CASE ABB OF
	0:
		IF mxEnable AND NOT CommData.mxABBExecuting THEN
			ABB:=10;
		END_IF
	10:
		IF CommData.mxRobotOnline THEN
			ABB:=100;
			ELSE
			ABB:=200;
		END_IF
	100:
		mxExecuting:=TRUE;
		CommData.maOrderMaker[1] := 2;
		CommData.maOrderMaker[2] := 0;
		CommData.maOrderMaker[3] := 0;
		CommData.maOrderMaker[4] := 0;
		CommData.maOrderMaker[5] := 0;
		CommData.maOrderMaker[6] := 0;
		CommData.qwOrderRobot:=200000;
		ABB:=101;
	101:
		IF CommData.qwOrderRobot > 0 THEN
			CommData.qxPLCStrobe:=TRUE;
			ABB:=102;
		END_IF
	102:
		IF CommData.ixRobotStrobe THEN
			IF CommData.iwReplyRobot = CommData.qwOrderRobot+1 THEN
				CommData.qwOrderRobot:=0;
				CommData.maOrderMaker[1] := 0;
				CommData.maOrderMaker[2] := 0;
				CommData.maOrderMaker[3] := 0;
				CommData.maOrderMaker[4] := 0;
				CommData.maOrderMaker[5] := 0;
				CommData.maOrderMaker[6] := 0;
				CommData.qxPLCStrobe:=FALSE;
				ABB:=103;
			ELSE
				ABB:=1000;
			END_IF
		END_IF
	103:
		IF NOT CommData.ixRobotStrobe THEN
			IF CommData.iwReplyRobot = 0 THEN
				ABB:=104;
			ELSE
				ABB:=1000;
			END_IF
		END_IF
	104:
		IF CommData.ixRobotStrobe THEN
			IF CommData.iwProgressRobot = 90 THEN
				CommData.qxPLCStrobe:=TRUE;
				ABB:=105;
			END_IF
			IF CommData.iwProgressRobot = 1000 THEN
				CommData.qxPLCStrobe:=TRUE;
				ABB:=1000;
			END_IF
		END_IF	
	105:
		IF  NOT CommData.ixRobotStrobe AND CommData.iwProgressRobot = 0 THEN
			CommData.qxPLCStrobe:=FALSE;
			ABB:=201;
		END_IF
		
	200:
		CommData.mwABBPosXaxis:=CommData.ABBPostions.AGVPOShome.X;
		CommData.mwABBPosYaxis:=CommData.ABBPostions.AGVPOShome.Y;
		mxExecuting:=TRUE;
		CommData.mxStartABB:=TRUE;
		IF CommData.mwXaxis = CommData.ABBPostions.AGVPOShome.X AND CommData.mwYaxis = CommData.ABBPostions.AGVPOShome.Y THEN
			ABB:=201;
		ELSIF gvl.ixEmergencyStop THEN
			ABB:=1000;
		END_IF
	201:
		mxExecuting:=FALSE;
		CommData.mxStartABB:=FALSE;
		mxDone:=TRUE;
		IF NOT mxEnable THEN
			mxDone:=FALSE;
			ABB:=0;
		END_IF
	1000:
		mxError:=TRUE;
		mxExecuting:=FALSE;
		CommData.mxStartABB:=FALSE;
		IF NOT mxEnable THEN
			mxError:=FALSE;
			mxDone:=FALSE;
			ABB:=0;
		END_IF
END_CASE



IF gvl.ixEmergencyStop THEN
	ABB:=1000;
END_IF

END_FUNCTION_BLOCK

// ---- ABBControl/ABBPickLeaveContainerAGV.TcPOU
FUNCTION_BLOCK ABBPickLeaveContainerAGV
VAR_INPUT
	mxEnable: BOOL;
	mxPick: BOOL;
END_VAR
VAR_OUTPUT
	mxDone:BOOL;
	mxExecuting: BOOL;
	mxError: BOOL;
END_VAR
VAR
	ABB: INT;
	mwordernumber: DINT;
END_VAR

CASE ABB OF
	0:
		IF mxEnable AND NOT CommData.mxABBExecuting THEN
			ABB:=10;
		END_IF
	10:
		IF CommData.mxRobotOnline THEN
			ABB:=100;
			ELSE
			ABB:=200;
		END_IF
	100:
		IF CommData.msRobotLastPos = 'AGV' THEN
			ABB:=101;
		ELSE
			ABB:=1000;
		END_IF
	101:
		mxExecuting:=TRUE;
		CommData.maOrderMaker[1] := 4;
		CommData.maOrderMaker[3] := 0;
		CommData.maOrderMaker[4] := 0;
		CommData.maOrderMaker[5] := 0;
		CommData.maOrderMaker[6] := 0;
		ABB:=102;
	102:
		IF mxPick THEN
			CommData.maOrderMaker[2] := 1;
			ABB:=103;
		ELSIF NOT mxPick THEN
			CommData.maOrderMaker[2] := 0;
			ABB:=103;
		END_IF
	103:
		mwordernumber:=CommData.maOrderMaker[1];
			mwordernumber:=mwordernumber*10;
			abb:=1151;
	1151:
			mwordernumber:=mwordernumber+CommData.maOrderMaker[2];
			abb:=1152;
	1152:
			mwordernumber:=mwordernumber*10;
			abb:=1153;
	1153:
			mwordernumber:=mwordernumber+CommData.maOrderMaker[3];
			abb:=1154;
	1154:
			mwordernumber:=mwordernumber*10;
			abb:=1155;
	1155:
			mwordernumber:=mwordernumber+CommData.maOrderMaker[4];
			abb:=1156;
	1156:
			mwordernumber:=mwordernumber*10;
			abb:=1157;
	1157:
			mwordernumber:=mwordernumber+CommData.maOrderMaker[5];
			abb:=1158;
	1158:
			mwordernumber:=mwordernumber*10;
			abb:=1159;
	1159:
			mwordernumber:=mwordernumber+CommData.maOrderMaker[6];
			ABB:=1160;
	1160:
		CommData.qwOrderRobot:=mwordernumber;
		ABB:=104;
	104:
		IF CommData.qwOrderRobot > 0 THEN
			CommData.qxPLCStrobe:=TRUE;
			ABB:=105;
		END_IF
	105:
		IF CommData.ixRobotStrobe THEN
			IF CommData.iwReplyRobot = CommData.qwOrderRobot+1 THEN
				CommData.qwOrderRobot:=0;
				mwordernumber:=0;
				CommData.qxPLCStrobe:=FALSE;
				ABB:=106;
			ELSE
				ABB:=1000;
			END_IF
		END_IF
	106:
		IF NOT CommData.ixRobotStrobe THEN
			IF CommData.iwReplyRobot = 0 THEN
				ABB:=107;
			ELSE
				ABB:=1000;
			END_IF
		END_IF
	107:
		IF CommData.ixRobotStrobe THEN
			IF CommData.iwProgressRobot = 90 THEN
				CommData.qxPLCStrobe:=TRUE;
				ABB:=108;
			END_IF
			IF CommData.iwProgressRobot = 1000 THEN
				CommData.qxPLCStrobe:=TRUE;
				ABB:=1000;
			END_IF
		END_IF
	108:
		IF  NOT CommData.ixRobotStrobe AND CommData.iwProgressRobot = 0 THEN
			CommData.qxPLCStrobe:=FALSE;
			ABB:=202;
		END_IF
		
		
		
	200:
		mxExecuting:=TRUE;
		IF CommData.mwXaxis = CommData.ABBPostions.AGVPOShome.X AND CommData.mwYaxis = CommData.ABBPostions.AGVPOShome.Y THEN
			ABB:=201;
		ELSE
			ABB:=1000;
		END_IF
	201:
		IF mxpick THEN
			IF NOT CommData.mxGripper THEN
				CommData.mxGripper:=TRUE;
				ABB:=202;
			ELSE
				ABB:=1000;
			END_IF
		ELSIF NOT mxPick THEN
			IF CommData.mxGripper THEN
				CommData.mxGripper:=FALSE;
				ABB:=202;
			ELSE
				ABB:=1000;
			END_IF
		END_IF
	202:
		mxExecuting:=FALSE;
		mxDone:=TRUE;
		IF NOT mxEnable THEN
			mxError:=FALSE;
			mxDone:=FALSE;
			ABB:=0;
		END_IF
	1000:
		mxError:=TRUE;
		mxExecuting:=FALSE;
		IF NOT mxEnable THEN
			mxError:=FALSE;
			mxDone:=FALSE;
			ABB:=0;
		END_IF
END_CASE





IF gvl.ixEmergencyStop THEN
	ABB:=1000;
END_IF

END_FUNCTION_BLOCK

// ---- ABBControl/ABBScanContainer.TcPOU
FUNCTION_BLOCK ABBScanContainer
VAR_INPUT
	mxEnable: BOOL;
	mwPartno: INT;
END_VAR
VAR_OUTPUT
	mxDone: BOOL;
	mxExecuting: BOOL;
	mxRobotatScanPos:BOOL;
	mxError: BOOL;
END_VAR
VAR
	ABB: INT;
	mxWaitingforsensorinput: BOOL;
	mwordernumber: DINT;
END_VAR

CASE ABB OF
		0:
			IF mxEnable AND NOT CommData.mxABBExecuting THEN
				ABB:=10;
			END_IF
		10:
			IF CommData.mxRobotOnline THEN
			ABB:=100;
			ELSE
			ABB:=200;
		END_IF
		100:
			IF CommData.msRobotLastPos = 'Table' THEN
				ABB:=101;
			ELSE
				ABB:=1000;
			END_IF
		101:
			mxExecuting:=TRUE;
			CommData.maOrderMaker[1] := 7;
			CommData.maOrderMaker[2] := 0;
			CommData.maOrderMaker[3] := 0;
			CommData.maOrderMaker[4] := 0;
			CommData.maOrderMaker[6] := 0;
			ABB:=102;
		102:
			IF mwPartno = 1 OR mwPartno = 2 OR mwPartno = 3 THEN
				CommData.maOrderMaker[5] := mwPartno;
				ABB:=103;
			ELSE
					ABB:=1000;//Error
			END_IF
		103:
			mwordernumber:=CommData.maOrderMaker[1];
				mwordernumber:=mwordernumber*10;
				abb:=1151;
		1151:
				mwordernumber:=mwordernumber+CommData.maOrderMaker[2];
				abb:=1152;
		1152:
			mwordernumber:=mwordernumber*10;
				abb:=1153;
		1153:
				mwordernumber:=mwordernumber+CommData.maOrderMaker[3];
				abb:=1154;
		1154:
				mwordernumber:=mwordernumber*10;
				abb:=1155;
		1155:
				mwordernumber:=mwordernumber+CommData.maOrderMaker[4];
				abb:=1156;
		1156:
				mwordernumber:=mwordernumber*10;
				abb:=1157;
		1157:
				mwordernumber:=mwordernumber+CommData.maOrderMaker[5];
				abb:=1158;
		1158:
				mwordernumber:=mwordernumber*10;
				abb:=1159;
		1159:
				mwordernumber:=mwordernumber+CommData.maOrderMaker[6];
				ABB:=1160;
		1160:
			CommData.qwOrderRobot:=mwordernumber;
			ABB:=104;
		104:
			IF CommData.qwOrderRobot > 0 THEN
				CommData.qxPLCStrobe:=TRUE;
				ABB:=105;
			END_IF
		105:
			IF CommData.ixRobotStrobe THEN
				IF CommData.iwReplyRobot = CommData.qwOrderRobot+1 THEN
					CommData.qwOrderRobot:=0;
					mwordernumber:=0;
					CommData.qxPLCStrobe:=FALSE;
					ABB:=106;
				ELSE
					ABB:=1000;
				END_IF
			END_IF
		106:
			IF NOT CommData.ixRobotStrobe THEN
				IF CommData.iwReplyRobot = 0 THEN
					ABB:=1061;
				ELSE
					ABB:=1000;
				END_IF
			END_IF
		1061:
			IF CommData.iwProgressRobot = 50 THEN
				mxRobotatScanPos:=TRUE;
				ABB:=107;
			END_IF
		107:
			IF CommData.ixRobotStrobe THEN
				mxRobotatScanPos:=FALSE;
				IF CommData.iwProgressRobot = 90 THEN
					CommData.qxPLCStrobe:=TRUE;
					ABB:=108;
				END_IF
				IF CommData.iwProgressRobot = 1000 THEN
					CommData.qxPLCStrobe:=TRUE;
					ABB:=1000;
				END_IF
			END_IF
		108:
			IF  NOT CommData.ixRobotStrobe AND CommData.iwProgressRobot = 0 THEN
				CommData.qxPLCStrobe:=FALSE;
				ABB:=203;
			END_IF
		
		
		
		
		
		200:
			IF mwPartno = 1 OR mwPartno = 2 OR mwPartno = 3 THEN
				ABB:=201;
			ELSE
				ABB:=1000;//Error
			END_IF
		201:
			IF CommData.mwXaxis = CommData.ABBPostions.Tablehome.X AND CommData.mwYaxis = CommData.ABBPostions.Tablehome.Y THEN
				ABB:=202;
			ELSE
				ABB:=1000;
			END_IF
		202:
			mxExecuting:=TRUE;
			mxRobotatScanPos:=TRUE;
			commdata.mxWaitingforSensorinput:=TRUE;
			IF GVL.ixInductiveSensorinTool OR CommData.mxScannernoobject THEN
				ABB:=203;
			END_IF
		203:
			commdata.mxWaitingforSensorinput:=FALSE;
			mxRobotatScanPos:=FALSE;
			mxExecuting:=FALSE;
			mxDone:=TRUE;
			IF NOT mxEnable THEN
				mxDone:=FALSE;
				ABB:=0;
			END_IF
		1000:
			mxExecuting:=FALSE;
			mxError:=TRUE;
			IF NOT mxEnable THEN
				mxError:=FALSE;
				mxDone:=FALSE;
				ABB:=0;
			END_IF
END_CASE



IF gvl.ixEmergencyStop THEN
	ABB:=1000;
END_IF

END_FUNCTION_BLOCK

// ---- ABBControl/ABBGotoTable.TcPOU
FUNCTION_BLOCK ABBGotoTable
VAR_INPUT
	mxEnable: BOOL;
END_VAR
VAR_OUTPUT
	mxDone:BOOL;
	mxExecuting: BOOL;
	mxError: BOOL;
END_VAR
VAR
	ABB: INT;
END_VAR

CASE ABB OF
	0:
		IF mxEnable AND NOT CommData.mxABBExecuting THEN
			ABB:=10;
		END_IF
	10:
		IF CommData.mxRobotOnline THEN
			ABB:=100;
		ELSE
			ABB:=200;
		END_IF
	100:
		mxExecuting:=TRUE;
		CommData.maOrderMaker[1] := 3;
		CommData.maOrderMaker[2] := 0;
		CommData.maOrderMaker[3] := 0;
		CommData.maOrderMaker[4] := 0;
		CommData.maOrderMaker[5] := 0;
		CommData.maOrderMaker[6] := 0;
		CommData.qwOrderRobot:=300000;
		ABB:=101;
	101:
		IF CommData.qwOrderRobot > 0 THEN
			CommData.qxPLCStrobe:=TRUE;
			ABB:=102;
		END_IF
	102:
		IF CommData.ixRobotStrobe THEN
			IF CommData.iwReplyRobot = CommData.qwOrderRobot+1 THEN
				CommData.qwOrderRobot:=0;
				CommData.maOrderMaker[1] := 0;
				CommData.maOrderMaker[2] := 0;
				CommData.maOrderMaker[3] := 0;
				CommData.maOrderMaker[4] := 0;
				CommData.maOrderMaker[5] := 0;
				CommData.maOrderMaker[6] := 0;
				CommData.qxPLCStrobe:=FALSE;
				ABB:=103;
			ELSE
				ABB:=1000;
			END_IF
		END_IF
	103:
		IF NOT CommData.ixRobotStrobe THEN
			IF CommData.iwReplyRobot = 0 THEN
				ABB:=104;
			ELSE
				ABB:=1000;
			END_IF
		END_IF
	104:
		IF CommData.ixRobotStrobe THEN
			IF CommData.iwProgressRobot = 90 THEN
				CommData.qxPLCStrobe:=TRUE;
				ABB:=105;
			END_IF
			IF CommData.iwProgressRobot = 1000 THEN
				CommData.qxPLCStrobe:=TRUE;
				ABB:=1000;
			END_IF
		END_IF	
	105:
		IF  NOT CommData.ixRobotStrobe AND CommData.iwProgressRobot = 0 THEN
			CommData.qxPLCStrobe:=FALSE;
			ABB:=201;
		END_IF
		
		
	200:
		CommData.mwABBPosXaxis:=CommData.ABBPostions.Tablehome.X;
		CommData.mwABBPosYaxis:=CommData.ABBPostions.Tablehome.Y;
		mxExecuting:=TRUE;
		CommData.mxStartABB:=TRUE;
		IF CommData.mwXaxis = CommData.ABBPostions.Tablehome.X AND CommData.mwYaxis = CommData.ABBPostions.Tablehome.Y THEN
			ABB:=201;
		ELSIF gvl.ixEmergencyStop THEN
			ABB:=1000;
		END_IF
	201:
		mxExecuting:=FALSE;
		CommData.mxStartABB:=FALSE;
		mxDone:=TRUE;
		IF NOT mxEnable THEN
			mxDone:=FALSE;
			ABB:=0;
		END_IF
	1000:
		mxError:=TRUE;
		mxExecuting:=FALSE;
		CommData.mxStartABB:=FALSE;
		IF NOT mxEnable THEN
			mxError:=FALSE;
			mxDone:=FALSE;
			ABB:=0;
		END_IF
END_CASE



IF gvl.ixEmergencyStop THEN
	ABB:=1000;
END_IF

END_FUNCTION_BLOCK

// ---- ABBControl/ABBAssemble.TcPOU
FUNCTION_BLOCK ABBAssemble
VAR_INPUT
	mxEnable: BOOL;
	mwBufferID: INT;
END_VAR
VAR_OUTPUT
	mxDone: BOOL;
	mxExecuting: BOOL;
	mxError: BOOL;
END_VAR
VAR
	ABB: INT;
	mwPlatecount: INT;
	mwordernumber: DINT;
END_VAR
VAR_INPUT
	mwAssemblePartno: INT;
END_VAR

CASE ABB OF
	0:
		IF mxEnable AND NOT CommData.mxABBExecuting THEN
			ABB:=10;
		END_IF
	10:
		IF CommData.mxRobotOnline THEN
			ABB:=11;
			ELSE
			ABB:=12;
		END_IF
	11:
		IF CommData.msRobotLastPos = 'Table' AND gvl.BufferProducts.Storage1.Quatity <> 0 AND gvl.BufferProducts.Storage2.Quatity <> 0 AND gvl.BufferProducts.Storage3.Quatity <> 0 THEN
			ABB:=111;
		ELSE
			ABB:=1000;
		END_IF
	111:
		mxExecuting:=TRUE;
		CommData.maOrderMaker[1] := 8;
		CommData.maOrderMaker[2] := 0;
		IF mwAssemblePartno =3 THEN
			abb:=112;
		ELSIF mwAssemblePartno =2 THEN
			abb:=113;
		ELSIF mwAssemblePartno =1 THEN
			abb:=114;
		END_IF	
	112:
		IF mwBufferID = 1 THEN
				CommData.maOrderMaker[3]:=mwBufferID;
				CommData.maOrderMaker[4]:=gvl.BufferProducts.Storage1.Quatity;
				CommData.maOrderMaker[5]:=mwAssemblePartno;
				CommData.maOrderMaker[6]:=0;
				abb:=115;
			ELSIF mwBufferID = 2 THEN
				CommData.maOrderMaker[3]:=mwBufferID;
				CommData.maOrderMaker[4]:=gvl.BufferProducts.Storage2.Quatity;
				CommData.maOrderMaker[5]:=mwAssemblePartno;
				CommData.maOrderMaker[6]:=0;
				abb:=115;
			ELSIF mwBufferID = 3 THEN
				CommData.maOrderMaker[3]:=mwBufferID;
				CommData.maOrderMaker[4]:=gvl.BufferProducts.Storage3.Quatity;
				CommData.maOrderMaker[5]:=mwAssemblePartno;
				CommData.maOrderMaker[6]:=0;
				abb:=115;
			ELSE
				ABB:=1000;
			END_IF
	113:
		IF mwBufferID = 1 THEN
				CommData.maOrderMaker[3]:=mwBufferID;
				CommData.maOrderMaker[4]:=gvl.BufferProducts.Storage1.Quatity;
				CommData.maOrderMaker[5]:=mwAssemblePartno;
				CommData.maOrderMaker[6]:=0;
				abb:=115;
			ELSIF mwBufferID = 2 THEN
				CommData.maOrderMaker[3]:=mwBufferID;
				CommData.maOrderMaker[4]:=gvl.BufferProducts.Storage2.Quatity;
				CommData.maOrderMaker[5]:=mwAssemblePartno;
				CommData.maOrderMaker[6]:=0;
				abb:=115;
			ELSIF mwBufferID = 3 THEN
				CommData.maOrderMaker[3]:=mwBufferID;
				CommData.maOrderMaker[4]:=gvl.BufferProducts.Storage3.Quatity;
				CommData.maOrderMaker[5]:=mwAssemblePartno;
				CommData.maOrderMaker[6]:=0;
				abb:=115;
			ELSE
				ABB:=1000;
			END_IF
	114:
		IF gvl.BufferProducts.Storage3.Quatity =2 THEN
			mwPlatecount:=6;
		ELSIF gvl.BufferProducts.Storage3.Quatity =1 THEN
			mwPlatecount:=5;
		END_IF
		IF mwBufferID = 1 THEN
				IF gvl.BufferProducts.Storage1.Quatity =2 THEN
					mwPlatecount:=6;
					abb:=1141;
				ELSIF gvl.BufferProducts.Storage1.Quatity =1 THEN
					mwPlatecount:=5;
					abb:=1141;
				END_IF
		ELSIF mwBufferID = 2 THEN
				IF gvl.BufferProducts.Storage2.Quatity =2 THEN
					mwPlatecount:=6;
					abb:=1141;
				ELSIF gvl.BufferProducts.Storage2.Quatity =1 THEN
					mwPlatecount:=5;
					abb:=1141;
				END_IF
		ELSIF mwBufferID = 3 THEN
				IF gvl.BufferProducts.Storage3.Quatity =2 THEN
					mwPlatecount:=6;
					abb:=1141;
				ELSIF gvl.BufferProducts.Storage3.Quatity =1 THEN
					mwPlatecount:=5;
					abb:=1141;
				END_IF
			ELSE
				ABB:=1000;
			END_IF
	1141:
		CommData.maOrderMaker[3]:=mwBufferID;
		CommData.maOrderMaker[4]:=mwPlatecount;
		CommData.maOrderMaker[5]:=mwAssemblePartno;
		CommData.maOrderMaker[6]:=0;
		abb:=115;
	115:
		IF CommData.maOrderMaker[1]=8 THEN
			mwordernumber:=CommData.maOrderMaker[1];
			mwordernumber:=mwordernumber*10;
			abb:=1151;
		END_IF
	1151:
			mwordernumber:=mwordernumber+CommData.maOrderMaker[2];
			abb:=1152;
	1152:
			mwordernumber:=mwordernumber*10;
			abb:=1153;
	1153:
			mwordernumber:=mwordernumber+CommData.maOrderMaker[3];
			abb:=1154;
	1154:
			mwordernumber:=mwordernumber*10;
			abb:=1155;
	1155:
			mwordernumber:=mwordernumber+CommData.maOrderMaker[4];
			abb:=1156;
	1156:
			mwordernumber:=mwordernumber*10;
			abb:=1157;
	1157:
			mwordernumber:=mwordernumber+CommData.maOrderMaker[5];
			abb:=1158;
	1158:
			mwordernumber:=mwordernumber*10;
			abb:=1159;
	1159:
			mwordernumber:=mwordernumber+CommData.maOrderMaker[6];
			ABB:=116;

	116:
		CommData.qwOrderRobot:=mwordernumber;
		ABB:=117;
	117:
		IF CommData.qwOrderRobot > 0 THEN
			CommData.qxPLCStrobe:=TRUE;
			ABB:=118;
		END_IF
	118:
		IF CommData.ixRobotStrobe THEN
			IF CommData.iwReplyRobot = CommData.qwOrderRobot+1 THEN
				CommData.qwOrderRobot:=0;
				mwordernumber:=0;
				CommData.qxPLCStrobe:=FALSE;
				ABB:=119;
			ELSE
				ABB:=1000;
			END_IF
		END_IF
	119:
		IF NOT CommData.ixRobotStrobe THEN
			IF CommData.iwReplyRobot = 0 THEN
				ABB:=120;
			ELSE
				ABB:=1000;
			END_IF
		END_IF
	120:
		IF CommData.ixRobotStrobe THEN
			IF CommData.iwProgressRobot = 90 THEN
				CommData.qxPLCStrobe:=TRUE;
				ABB:=121;
			END_IF
			IF CommData.iwProgressRobot = 1000 THEN
				CommData.qxPLCStrobe:=TRUE;
				ABB:=1000;
			END_IF
		END_IF
	121:
		IF  NOT CommData.ixRobotStrobe AND CommData.iwProgressRobot = 0 THEN
			CommData.qxPLCStrobe:=FALSE;
			ABB:=73;
		END_IF
	12:
		IF CommData.mwXaxis = CommData.ABBPostions.Tablehome.X AND CommData.mwYaxis = CommData.ABBPostions.Tablehome.Y THEN
			ABB:=20;
		ELSE
			ABB:=1000;
		END_IF
	20:
		mxExecuting:=TRUE;
		CommData.mwABBPosXaxis:=CommData.ABBPostions.Bufferhome.X;
		CommData.mwABBPosYaxis:=CommData.ABBPostions.Bufferhome.Y;
		CommData.mxStartABB:=TRUE;
		IF CommData.mwXaxis = CommData.ABBPostions.Bufferhome.X AND CommData.mwYaxis = CommData.ABBPostions.Bufferhome.Y THEN
			CommData.mxStartABB:=FALSE;
			ABB:=30;
		ELSIF gvl.ixEmergencyStop THEN
			ABB:=1000;
		END_IF
	30:
		IF mwBufferID = 1 THEN
			ABB:=40;
		ELSIF mwBufferID = 2 THEN
			ABB:=50;
		ELSIF mwBufferID = 3 THEN
			ABB:=60;
		ELSE
			ABB:=1000;//Error
		END_IF
	40:
		CommData.mwABBPosXaxis:=CommData.ABBPostions.Storage1.X;
		CommData.mwABBPosYaxis:=CommData.ABBPostions.Storage1.Y;
		CommData.mxStartABB:=TRUE;
		IF CommData.mwXaxis = CommData.ABBPostions.Storage1.X AND CommData.mwYaxis = CommData.ABBPostions.Storage1.Y THEN
			CommData.mxStartABB:=FALSE;
			ABB:=70;
		END_IF
	50:
		CommData.mwABBPosXaxis:=CommData.ABBPostions.Storage2.X;
		CommData.mwABBPosYaxis:=CommData.ABBPostions.Storage2.Y;
		CommData.mxStartABB:=TRUE;
		IF CommData.mwXaxis = CommData.ABBPostions.Storage2.X AND CommData.mwYaxis = CommData.ABBPostions.Storage2.Y THEN
			CommData.mxStartABB:=FALSE;
			ABB:=70;
		END_IF
	60:
		CommData.mwABBPosXaxis:=CommData.ABBPostions.Storage3.X;
		CommData.mwABBPosYaxis:=CommData.ABBPostions.Storage3.Y;
		CommData.mxStartABB:=TRUE;
		IF CommData.mwXaxis = CommData.ABBPostions.Storage3.X AND CommData.mwYaxis = CommData.ABBPostions.Storage3.Y THEN
			CommData.mxStartABB:=FALSE;
			ABB:=70;
		END_IF
		
		
		
	70:
		IF NOT CommData.mxABBExecuting THEN
			IF NOT CommData.mxGripper THEN
				CommData.mxGripper:=TRUE;
				ABB:=71;
			ELSE
				ABB:=1000;
			END_IF
		END_IF
	71:
		CommData.mwABBPosXaxis:=CommData.ABBPostions.Tablehome.X;
		CommData.mwABBPosYaxis:=CommData.ABBPostions.Tablehome.Y;
		CommData.mxStartABB:=TRUE;
		IF CommData.mwXaxis = CommData.ABBPostions.Tablehome.X AND CommData.mwYaxis = CommData.ABBPostions.Tablehome.Y THEN
			CommData.mxStartABB:=FALSE;
			ABB:=72;
		END_IF
	72:
		IF CommData.mxGripper THEN
			CommData.mxGripper:=FALSE;
			ABB:=73;
		ELSE
			ABB:=40;
		END_IF
	73:
		mxExecuting:=FALSE;
		mxDone:=TRUE;
		IF NOT mxEnable THEN
			mxError:=FALSE;
			mxDone:=FALSE;
			ABB:=0;
		END_IF
	1000:
		mxError:=TRUE;
		mxExecuting:=FALSE;
		CommData.mxStartABB:=FALSE;
		IF NOT mxEnable THEN
			mxError:=FALSE;
			mxDone:=FALSE;
			ABB:=0;
		END_IF
END_CASE


IF gvl.ixEmergencyStop THEN
	ABB:=1000;
END_IF

END_FUNCTION_BLOCK

// ---- ABBControl/ABBPickLeaveContaineronTable.TcPOU
FUNCTION_BLOCK ABBPickLeaveContaineronTable
VAR_INPUT
	mxEnable: BOOL;
	mxPick: BOOL;
END_VAR
VAR_OUTPUT
	mxDone:BOOL;
	mxExecuting: BOOL;
	mxError: BOOL;
END_VAR
VAR
	ABB: INT;
	mwordernumber: DINT;
END_VAR

CASE ABB OF
	0:
		IF mxEnable AND NOT CommData.mxABBExecuting THEN
			ABB:=10;
		END_IF
	10:
		IF CommData.mxRobotOnline THEN
			ABB:=100;
			ELSE
			ABB:=200;
		END_IF
	100:
		IF CommData.msRobotLastPos = 'Table' THEN
			ABB:=101;
		ELSE
			ABB:=1000;
		END_IF
	101:
		mxExecuting:=TRUE;
		CommData.maOrderMaker[1] := 5;
		CommData.maOrderMaker[3] := 0;
		CommData.maOrderMaker[4] := 0;
		CommData.maOrderMaker[5] := 0;
		CommData.maOrderMaker[6] := 0;
		ABB:=102;
	102:
		IF mxPick THEN
			CommData.maOrderMaker[2] := 1;
			ABB:=103;
		ELSIF NOT mxPick THEN
			CommData.maOrderMaker[2] := 0;
			ABB:=103;
		END_IF
	103:
		mwordernumber:=CommData.maOrderMaker[1];
			mwordernumber:=mwordernumber*10;
			abb:=1151;
	1151:
			mwordernumber:=mwordernumber+CommData.maOrderMaker[2];
			abb:=1152;
	1152:
			mwordernumber:=mwordernumber*10;
			abb:=1153;
	1153:
			mwordernumber:=mwordernumber+CommData.maOrderMaker[3];
			abb:=1154;
	1154:
			mwordernumber:=mwordernumber*10;
			abb:=1155;
	1155:
			mwordernumber:=mwordernumber+CommData.maOrderMaker[4];
			abb:=1156;
	1156:
			mwordernumber:=mwordernumber*10;
			abb:=1157;
	1157:
			mwordernumber:=mwordernumber+CommData.maOrderMaker[5];
			abb:=1158;
	1158:
			mwordernumber:=mwordernumber*10;
			abb:=1159;
	1159:
			mwordernumber:=mwordernumber+CommData.maOrderMaker[6];
			ABB:=1160;
	1160:
		CommData.qwOrderRobot:=mwordernumber;
		ABB:=104;
	104:
		IF CommData.qwOrderRobot > 0 THEN
			CommData.qxPLCStrobe:=TRUE;
			ABB:=105;
		END_IF
	105:
		IF CommData.ixRobotStrobe THEN
			IF CommData.iwReplyRobot = CommData.qwOrderRobot+1 THEN
				CommData.qwOrderRobot:=0;
				mwordernumber:=0;
				CommData.qxPLCStrobe:=FALSE;
				ABB:=106;
			ELSE
				ABB:=1000;
			END_IF
		END_IF
	106:
		IF NOT CommData.ixRobotStrobe THEN
			IF CommData.iwReplyRobot = 0 THEN
				ABB:=107;
			ELSE
				ABB:=1000;
			END_IF
		END_IF
	107:
		IF CommData.ixRobotStrobe THEN
			IF CommData.iwProgressRobot = 90 THEN
				CommData.qxPLCStrobe:=TRUE;
				ABB:=108;
			END_IF
			IF CommData.iwProgressRobot = 1000 THEN
				CommData.qxPLCStrobe:=TRUE;
				ABB:=1000;
			END_IF
		END_IF
	108:
		IF  NOT CommData.ixRobotStrobe AND CommData.iwProgressRobot = 0 THEN
			CommData.qxPLCStrobe:=FALSE;
			ABB:=202;
		END_IF
	

	200:
		mxExecuting:=TRUE;
		IF CommData.mwXaxis = CommData.ABBPostions.Tablehome.X AND CommData.mwYaxis = CommData.ABBPostions.Tablehome.Y THEN
			ABB:=201;
		ELSE
			mxError:=TRUE;
			ABB:=40;
		END_IF
	201:
		IF mxpick THEN
			IF NOT CommData.mxGripper THEN
				CommData.mxGripper:=TRUE;
				ABB:=202;
			ELSE
				ABB:=1000;
			END_IF
		ELSIF NOT mxPick THEN
			IF CommData.mxGripper THEN
				CommData.mxGripper:=FALSE;
				ABB:=202;
			ELSE
				ABB:=1000;
			END_IF
		END_IF
	202:
		mxExecuting:=FALSE;
		mxDone:=TRUE;
		IF NOT mxEnable THEN
			mxError:=FALSE;
			mxDone:=FALSE;
			ABB:=0;
		END_IF
	1000:  //Error State
		mxError:=TRUE;
		mxExecuting:=FALSE;
		IF NOT mxEnable THEN
			mxError:=FALSE;
			mxDone:=FALSE;
			ABB:=0;
		END_IF
END_CASE




IF gvl.ixEmergencyStop THEN
	ABB:=1000;
END_IF

END_FUNCTION_BLOCK

// ---- Automation Library/PhysicalSystemTest.TcPOU
PROGRAM PhysicalSystemTest
VAR
	ABB: INT;
	TwoSecTimer: TON;
	mxTimerStart:BOOL;
	mxTimerDone:BOOL;
END_VAR

CASE ABB OF
	0:
		IF CommData.qxPLCStrobe THEN
			ABB:=10;
		END_IF
	10:
		IF CommData.qwOrderRobot > 0 THEN
			CommData.iwReplyRobot:=CommData.qwOrderRobot+1;
			mxTimerStart:=TRUE;
			ABB:=20;
		END_IF
	20:
		IF mxTimerDone THEN
			CommData.ixRobotStrobe :=TRUE;
			mxTimerStart:=FALSE;
			ABB:=30;
		END_IF
	30:
		IF NOT CommData.qxPLCStrobe THEN
			mxTimerStart:=TRUE;
			ABB:=40;
		END_IF
	40:
		IF mxTimerDone THEN
			CommData.iwReplyRobot:=0;
			CommData.ixRobotStrobe :=FALSE;
			mxTimerStart:=FALSE;
			ABB:=50;
		END_IF
	50:
		mxTimerStart:=TRUE;
		IF mxTimerDone THEN
			mxTimerStart:=FALSE;
			CommData.iwProgressRobot:=90;
			ABB:=60;
		END_IF
	60:
		CommData.ixRobotStrobe :=TRUE;
		mxTimerStart:=TRUE;
		ABB:=70;
	70:
		IF mxTimerDone AND CommData.qxPLCStrobe THEN
			mxTimerStart:=FALSE;
			CommData.iwProgressRobot:=0;
			ABB:=80;
		END_IF
	80:
		mxTimerStart:=TRUE;
		IF mxTimerDone THEN
			mxTimerStart:=FALSE;
			CommData.ixRobotStrobe :=FALSE;
			ABB:=90;
		END_IF
	90:
		IF NOT CommData.qxPLCStrobe THEN
			ABB:=0;
		END_IF
END_CASE



TwoSecTimer(IN:= mxTimerStart, PT:= T#2S, Q=> mxTimerDone, ET=> );

END_PROGRAM

// ---- GlobalTextList.TcGTLO
TEXTLIST GlobalTextList
  153 = ' %s'
  135 = '%s'
  875 = '1'
  207 = '2'
  288 = '3'
  990 = 'ABB Error'
  910 = 'ABB Executing'
  564 = 'ABB Functions'
  615 = 'ABB Onlibe'
  693 = 'ABB Status'
  435 = 'AGV'
  139 = 'AGV at Station :'
  241 = 'AGV Pos'
  375 = 'AGV Scan Table'
  171 = 'All Buffer Check'
  575 = 'All Home Check'
  974 = 'Aseembly'
  126 = 'Assemble'
  522 = 'Assembling'
  423 = 'Auto'
  27 = 'Auto Mode'
  641 = 'Booking from IO Station  :'
  114 = 'Buffer'
  731 = 'Buffer 1'
  938 = 'Buffer 2'
  402 = 'Buffer 3'
  289 = 'Buffer Empty'
  769 = 'Buffer ID'
  25 = 'BufferID'
  512 = 'Checkbox'
  728 = 'Container'
  514 = 'Container Color'
  281 = 'Control for Station'
  685 = 'Cylinder'
  150 = 'Debug Mode'
  228 = 'DebugMode'
  379 = 'Dummy BUffer'
  698 = 'Dummy Buffer'
  390 = 'Emergency Mode'
  137 = 'Emergency Signal :'
  493 = 'Emergency Stop'
  136 = 'Error from Comm :'
  999 = 'Execute'
  93 = 'Finish Order'
  170 = 'Gabriel Sebastian'
  751 = 'Gabriel Sebastian gabriel.sebastian@hv.se'
  995 = 'Gabriel Sebastian | gabriel.sebastian@hv.se'
  701 = 'Gabriel Sebastian |gabriel.sebastian@hv.se'
  922 = 'Go to Pos'
  688 = 'Gripper Control'
  247 = 'Gripper Toggle'
  222 = 'Home'
  140 = 'Inventory Status'
  395 = 'ixAGVatStation'
  884 = 'Leave'
  498 = 'Leave at AGV'
  298 = 'Main Menu'
  319 = 'Manual'
  917 = 'Manual Controller'
  314 = 'Manual Controls'
  212 = 'Manual Mode'
  122 = 'Manual Scanning'
  792 = 'Mode Status'
  1015 = 'New AGV to Station'
  203 = 'New AGV to Station :'
  151 = 'Normal Mode'
  908 = 'Octagon'
  287 = 'OFF'
  363 = 'Offline'
  741 = 'OFFLINE'
  374 = 'ON'
  13 = 'Online'
  979 = 'ONLINE'
  174 = 'Order for Next Assembly  : %s'
  138 = 'Pallet Placed on AGV :'
  147 = 'Pallet Sensor 1  :'
  146 = 'Pallet Sensor 2  :'
  148 = 'Pallet Sensor 3  :'
  145 = 'Pallet Sensor 4  :'
  563 = 'Part'
  315 = 'Part 1'
  242 = 'Part 2'
  436 = 'Part 3'
  331 = 'Part ID'
  213 = 'PartID'
  874 = 'Pause'
  105 = 'Paused'
  339 = 'Pick'
  758 = 'Pick / Leave'
  110 = 'Plate'
  669 = 'PLC'
  646 = 'Quantity'
  196 = 'Request Generator'
  835 = 'Reset'
  166 = 'Reset ABB'
  883 = 'Reset Station'
  867 = 'Reset Task'
  556 = 'Robot'
  625 = 'Robot Position  : %s'
  881 = 'Robot Power'
  502 = 'Robot Station'
  583 = 'Scan Buffer 1'
  714 = 'Scan Buffer 2'
  354 = 'Scan Buffer 3'
  620 = 'Scan Container'
  204 = 'Scanner'
  973 = 'Scanning'
  83 = 'Send Order'
  899 = 'Sensor Reading  : %s'
  238 = 'Sensor Reading completed'
  144 = 'Sensor Signals'
  134 = 'Station ID :'
  152 = 'Station Offline'
  494 = 'Station Status  : %s'
  458 = 'Station View'
  169 = 'Stop'
  143 = 'Storage Pos 1: %s'
  141 = 'Storage Pos 2: %s'
  142 = 'Storage Pos 3: %s'
  456 = 'SubTask'
  549 = 'Table'
  266 = 'Table To AGV'
  882 = 'Task'
  229 = 'Task Section'
  309 = 'Test System'
  149 = 'Tool Sensor  :'
  886 = 'Visualization'
  127 = 'X  : %s'
  412 = 'Y  : %s'
END_TEXTLIST

// ---- VISUs/RobotStation.TcVIS
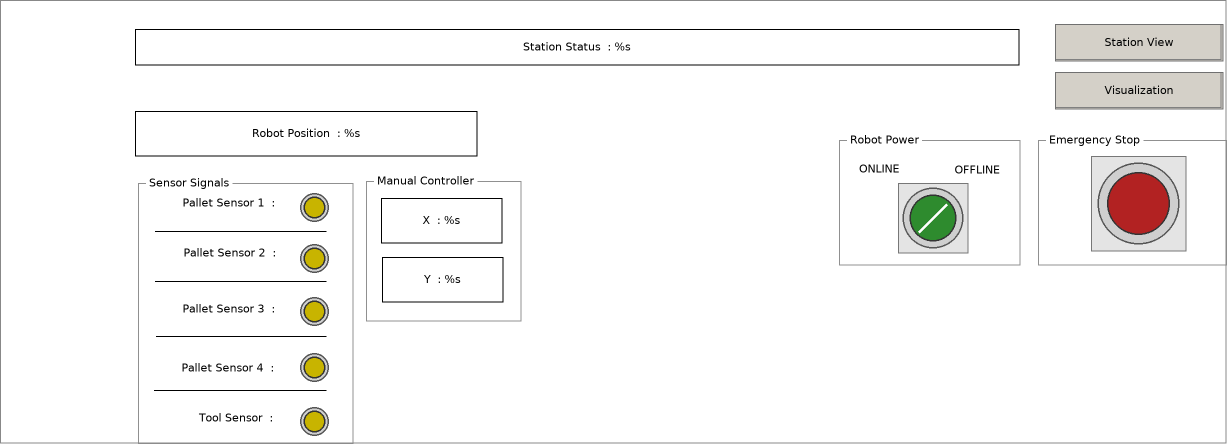
VISUALIZATION RobotStation  // 1227x444
    Rectangle (135,29 884x36), "Station Status : %s", text variable: Visualaisation_Control.mxStationStatus
    GroupBox (839,132 181x133), "Robot Power", invisible if: CommData.mxOnlineMode
        RotarySwitch (59,51 70x70), variable: CommData.mxRobotOnline, invisible if: CommData.mxOnlineMode, behaviour: TOGGLE, style: Switch-RotarySwitch-Green
        Label (11,22 59x30), "ONLINE"
        Label (106,23 65x30), "OFFLINE"
    Button (1055,72 168x37), "Visualization"
        OnMouseClick: change screen: Visualization
    GroupBox (1038,132 189x133), "Emergency Stop"
        PushSwitch (45,24 111x95), variable: GVL.ixEmergencyStop, behaviour: TOGGLE, style: Switch-PushSwitch-Red
    Rectangle (135,111 342x45), "Robot Position : %s", text variable: CommData.msRobotLastPos
    GroupBox (138,175 215x269), "Sensor Signals"
        Label (15,178 150x30), "Pallet Sensor 4 :"
        Label (17,63 150x30), "Pallet Sensor 2 :"
        Line (17,56) (188,56)
        Lamp1 (160,16 33x33), variable: GVL.ixInductiveSensor1, style: Lamp-Lamp1-Yellow
        Lamp1 (160,67 33x33), variable: GVL.ixInductiveSensor2, style: Lamp-Lamp1-Yellow
        Lamp1 (160,120 33x33), variable: GVL.ixInductiveSensor3, style: Lamp-Lamp1-Yellow
        Lamp1 (160,176 33x33), variable: GVL.ixInductiveSensor4, style: Lamp-Lamp1-Yellow
        Label (16,119 150x30), "Pallet Sensor 3 :"
        Label (23,228 150x30), "Tool Sensor :"
        Lamp1 (160,230 33x33), variable: GVL.ixInductiveSensorinTool, style: Lamp-Lamp1-Yellow
        Line (17,106) (188,106)
        Line (18,161) (188,161)
        Line (16,215) (188,215)
        Label (16,13 150x30), "Pallet Sensor 1 :"
    GroupBox (366,173 155x148), "Manual Controller"
        Rectangle (16,84 121x45), "Y : %s", text variable: CommData.mwYaxis
            OnMouseClick: write the text variable via Default
        Rectangle (15,25 121x45), "X : %s", text variable: CommData.mwXaxis
            OnMouseClick: write the text variable via Default
    Button (1055,24 168x37), "Station View"
        OnMouseClick: change screen: Station
END_VISUALIZATION

// ---- VISUs/Station.TcVIS
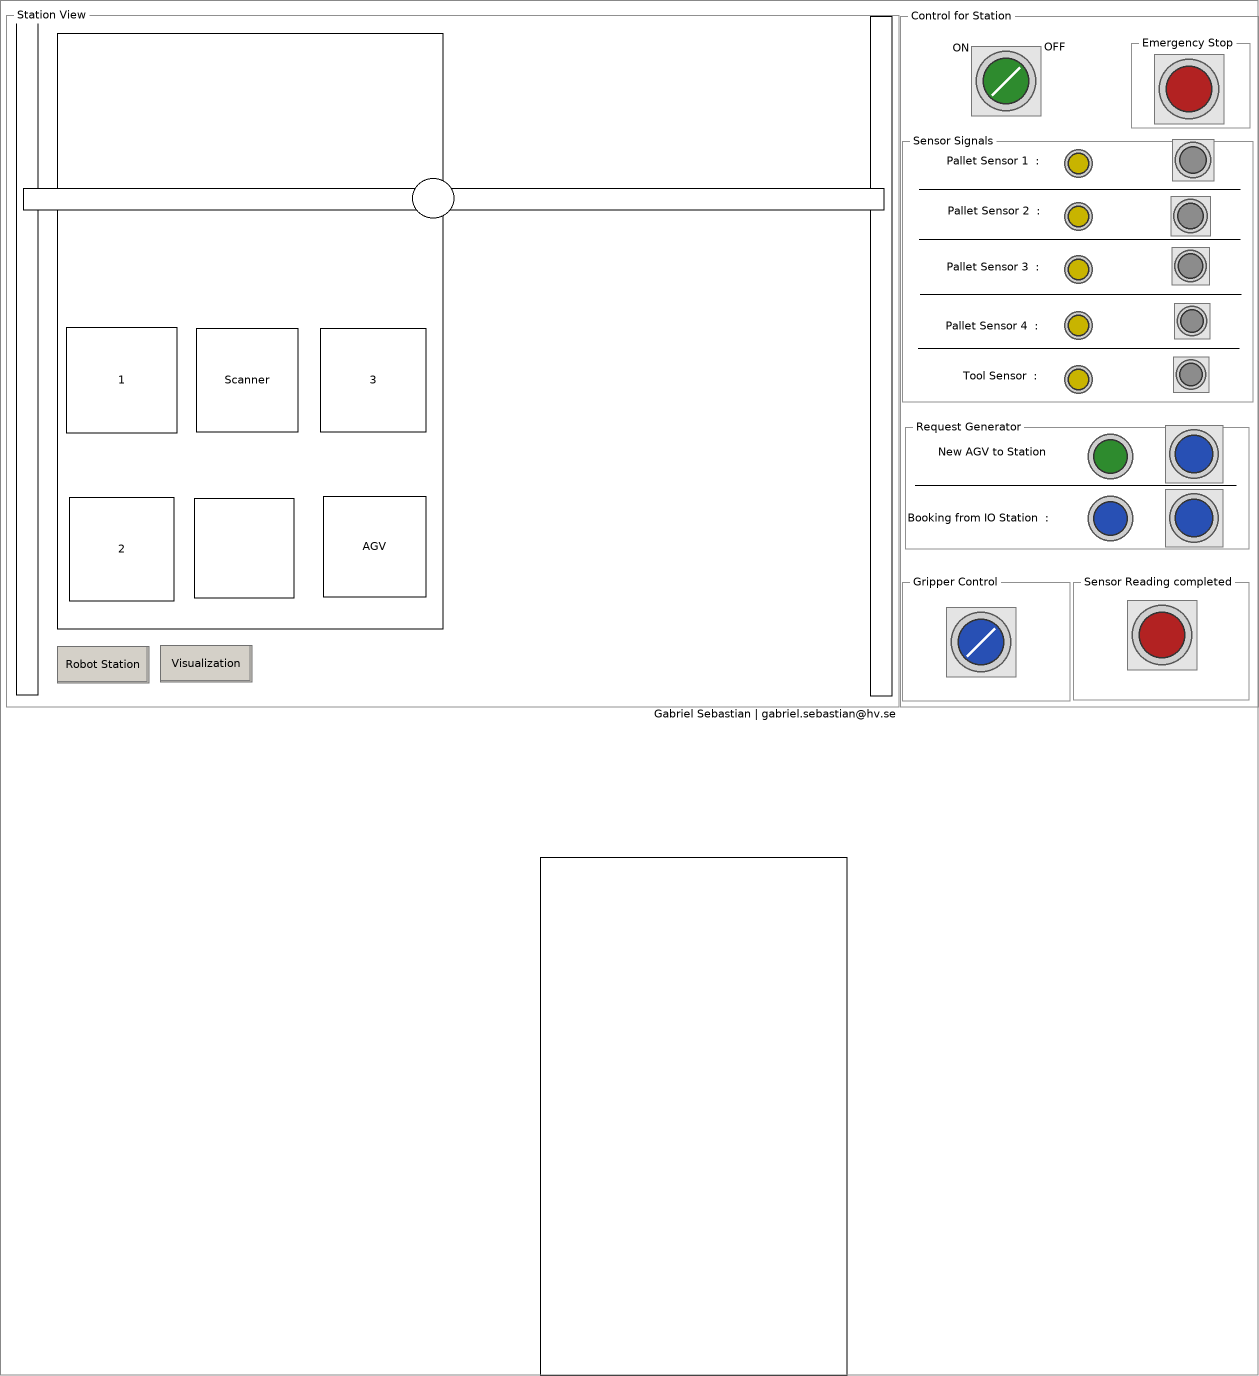
VISUALIZATION Station  // 1259x1376
    RoundedRectangle (540,857 307x519)
        p2738717112: CommData.mwCurrentAGVPOS
    Rectangle (16,15 22x680)
    GroupBox (6,7 893x700), "Station View"
        Rectangle (51,26 386x596)
        Rectangle (864,9 22x680)
        Rectangle (188,491 100x100)
        Rectangle (317,489 103x101), "AGV"
        Rectangle (190,321 102x104), "Scanner"
        Rectangle (60,320 111x106), "1"
        Rectangle (314,321 106x104), "3"
        Rectangle (63,490 105x104), "2"
        RoundedRectangle (17,181 861x22)
            p2738717112: CommData.mwYaxis
        Ellipse (406,171 42x40)
            p2738717112: CommData.mwYaxis
            p3560616238: CommData.mwXaxis
        Button (154,638 92x37), "Visualization"
            OnMouseClick: change screen: Visualization
        Button (51,639 92x37), "Robot Station"
            OnMouseClick: change screen: RobotStation
    GroupBox (900,8 359x699), "Control for Station"
        GroupBox (2,125 351x269), "Sensor Signals"
            Label (15,178 150x30), "Pallet Sensor 4 :"
            Label (17,63 150x30), "Pallet Sensor 2 :"
            Label (16,13 150x30), "Pallet Sensor 1 :"
            Line (17,56) (338,56)
            Lamp1 (160,14 33x33), variable: GVL.ixInductiveSensor1, style: Lamp-Lamp1-Yellow
            Lamp1 (160,67 33x33), variable: GVL.ixInductiveSensor2, style: Lamp-Lamp1-Yellow
            Lamp1 (160,120 33x33), variable: GVL.ixInductiveSensor3, style: Lamp-Lamp1-Yellow
            Lamp1 (160,176 33x33), variable: GVL.ixInductiveSensor4, style: Lamp-Lamp1-Yellow
            Label (16,119 150x30), "Pallet Sensor 3 :"
            Label (23,228 150x30), "Tool Sensor :"
            Lamp1 (160,230 33x33), variable: GVL.ixInductiveSensorinTool, style: Lamp-Lamp1-Yellow
            PushSwitch (266,6 50x42), variable: GVL.ixInductiveSensor1, input disabled if: CommData.mxRobotOnline, behaviour: TOGGLE, style: Switch-PushSwitch-Gray
            PushSwitch (267,63 43x40), variable: GVL.ixInductiveSensor2, input disabled if: CommData.mxRobotOnline, behaviour: TOGGLE, style: Switch-PushSwitch-Gray
            PushSwitch (269,114 39x38), variable: GVL.ixInductiveSensor3, input disabled if: CommData.mxRobotOnline, behaviour: TOGGLE, style: Switch-PushSwitch-Gray
            PushSwitch (270,170 40x36), variable: GVL.ixInductiveSensor4, input disabled if: CommData.mxRobotOnline, behaviour: TOGGLE, style: Switch-PushSwitch-Gray
            PushSwitch (271,223 36x37), variable: GVL.ixInductiveSensorinTool, input disabled if: CommData.mxRobotOnline, behaviour: TOGGLE, style: Switch-PushSwitch-Gray
            Line (17,106) (338,106)
            Line (18,161) (339,161)
            Line (16,215) (337,215)
        RotarySwitch (71,38 70x70), variable: CommData.mxOnlineMode, invisible if: CommData.mxRobotOnline, behaviour: TOGGLE, style: Switch-RotarySwitch-Green
        Label (106,24 98x30), "OFF", invisible if: CommData.mxRobotOnline
        Label (12,25 98x30), "ON", invisible if: CommData.mxRobotOnline
        GroupBox (5,411 344x130), "Request Generator"
            Label (12,18 150x30), "New AGV to Station"
            Line (10,66) (331,66)
            Lamp1 (177,11 57x53), variable: GVL.ixAGVatStation, style: Lamp-Lamp1-Green
            Lamp1 (177,73 57x53), variable: CommData.mxNewBookingrequest, style: Lamp-Lamp1-Blue
            PushSwitch (259,70 60x58), variable: CommData.mxNewBookingrequest, behaviour: TOGGLE, style: Switch-PushSwitch-Blue
        GroupBox (173,566 176x126), "Sensor Reading completed", invisible if: NOT CommData.mxWaitingforSensorinput
            PushSwitch (54,26 70x70), variable: CommData.mxScannernoobject, behaviour: TAP, style: Switch-PushSwitch-Red
        GroupBox (2,566 168x127), "Gripper Control"
            Lamp1 (-1748,-553 70x70), style: Lamp-Lamp1-Yellow
            Lamp1 (44,34 70x70), variable: CommData.mxGripper, style: Lamp-Lamp1-Yellow
            RotarySwitch (44,33 70x70), variable: CommData.mxGripper, invisible if: NOT Visualaisation_Control.mxManualMode, behaviour: TOGGLE, style: Switch-RotarySwitch-Blue
        GroupBox (231,27 119x93), "Emergency Stop"
            PushSwitch (23,19 70x70), variable: GVL.ixEmergencyStop, behaviour: TOGGLE, style: Switch-PushSwitch-Red
    Label (900,503 156x30), "Booking from IO Station :"
    Label (650,699 250x30), "Gabriel Sebastian | gabriel.sebastian@hv.se"
    PushSwitch (1164,425 60x58), variable: CommData.mxRequestAGV, behaviour: TOGGLE, style: Switch-PushSwitch-Blue
END_VISUALIZATION

// ---- VISUs/Visualization.TcVIS
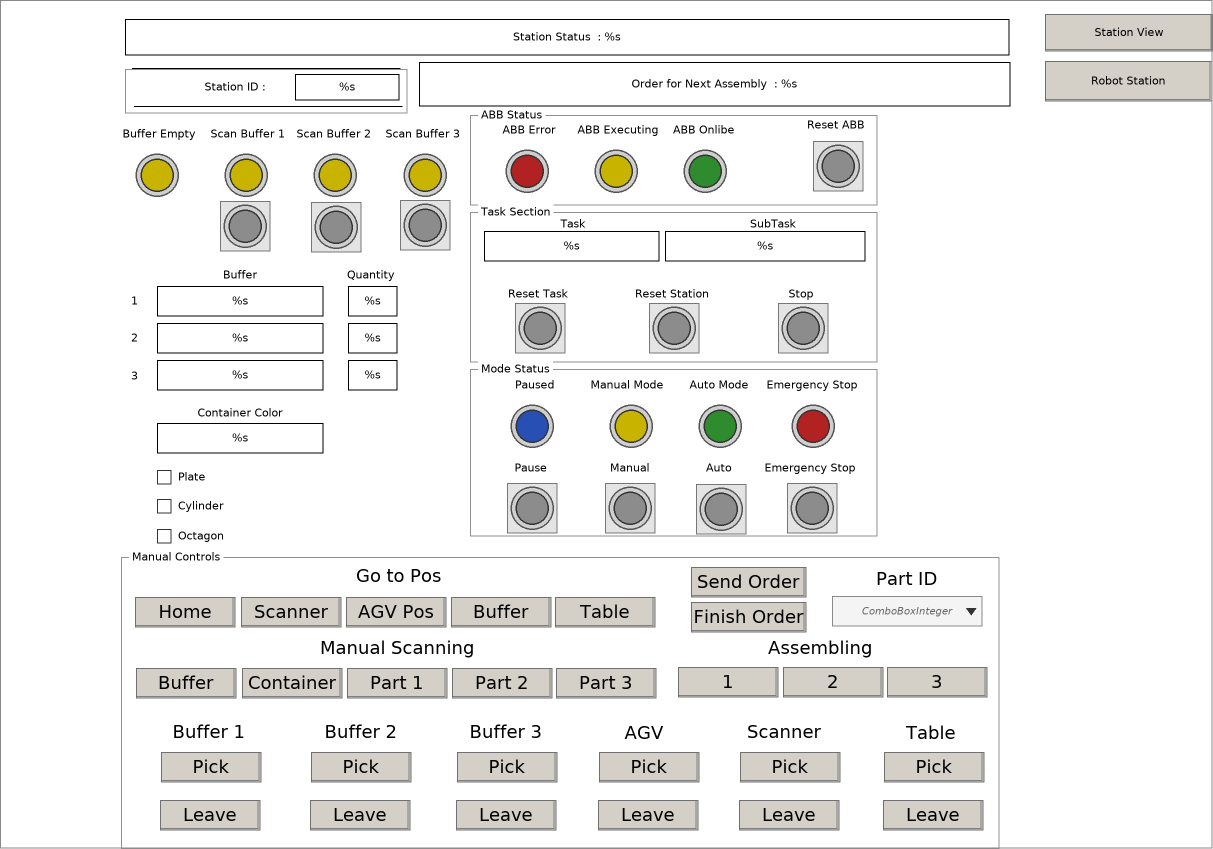
VISUALIZATION Visualization  // 1213x849
    Rectangle (125,19 884x36), "Station Status : %s", text variable: Visualaisation_Control.mxStationStatus
    GroupBox (125,61 282x52)
        Line (7,7) (275,7)
        Label (35,11 150x30), "Station ID :"
        Rectangle (170,13 104x26), "%s", text variable: GVL.mwStationID
        Line (9,45) (277,45)
    Button (1045,61 167x40), "Robot Station"
        OnMouseClick: change screen: RobotStation
    Rectangle (419,62 591x44), "Order for Next Assembly : %s", text variable: GVL.qsOrderFornextAssembly
    Button (1045,14 168x37), "Station View"
        OnMouseClick: change screen: Station
    Lamp1 (132,150 50x50), variable: MAIN.ixEmptyBuffer, style: Lamp-Lamp1-Yellow
    Label (84,119 150x30), "Buffer Empty"
    Lamp1 (221,150 50x50), style: Lamp-Lamp1-Yellow
    Label (173,119 150x30), "Scan Buffer 1"
    Lamp1 (310,150 50x50), style: Lamp-Lamp1-Yellow
    Label (259,119 150x30), "Scan Buffer 2"
    Lamp1 (400,150 50x50), style: Lamp-Lamp1-Yellow
    Label (348,119 150x30), "Scan Buffer 3"
    GroupBox (470,107 407x98), "ABB Status"
        PushSwitch (343,34 50x50), variable: MAIN.ixResetABB, behaviour: TAP, style: Switch-PushSwitch-Gray
        Label (291,3 150x30), "Reset ABB"
    Lamp1 (502,146 50x50), variable: MAIN.qxABBErrorLamp, style: Lamp-Lamp1-Red
    Label (454,115 150x30), "ABB Error"
    Lamp1 (591,146 50x50), variable: MAIN.qxABBExecutLamp, style: Lamp-Lamp1-Yellow
    Label (543,115 150x30), "ABB Executing"
    Lamp1 (680,146 50x50), variable: MAIN.qxABBonlineLamp, style: Lamp-Lamp1-Green
    Label (629,115 150x30), "ABB Onlibe"
    GroupBox (470,204 407x158), "Task Section"
        Rectangle (14,27 175x30), "%s", text variable: MAIN.qsTask
        Rectangle (195,27 200x30), "%s", text variable: MAIN.qsSubTask
        PushSwitch (179,99 50x50), behaviour: TAP, style: Switch-PushSwitch-Gray
        PushSwitch (308,99 50x50), behaviour: TAP, style: Switch-PushSwitch-Gray
    Label (498,209 150x30), "Task"
    Label (698,209 150x30), "SubTask"
    PushSwitch (515,303 50x50), behaviour: TAP, style: Switch-PushSwitch-Gray
    Label (463,279 150x30), "Reset Task"
    Label (597,279 150x30), "Reset Station"
    Label (726,279 150x30), "Stop"
    GroupBox (470,361 407x175), "Mode Status"
        PushSwitch (37,122 50x50), variable: MAIN.ixPauseButt, behaviour: TOGGLE, style: Switch-PushSwitch-Gray
        PushSwitch (135,122 50x50), variable: MAIN.qxManualMode, behaviour: TAP, style: Switch-PushSwitch-Gray
        PushSwitch (226,123 50x50), variable: MAIN.qxAutoMode, behaviour: TAP, style: Switch-PushSwitch-Gray
        PushSwitch (317,122 50x50), variable: GVL.ixEmergencyStop, behaviour: TOGGLE, style: Switch-PushSwitch-Gray
        Label (174,92 150x30), "Auto"
        Label (265,92 150x30), "Emergency Stop"
    Lamp1 (507,401 50x50), variable: MAIN.qxPauseLamp, style: Lamp-Lamp1-Blue
    Label (460,370 150x30), "Paused"
    Lamp1 (606,401 50x50), variable: MAIN.ixManualLamp, style: Lamp-Lamp1-Yellow
    Label (552,370 150x30), "Manual Mode"
    Lamp1 (695,401 50x50), variable: MAIN.ixAutoLamp, style: Lamp-Lamp1-Green
    Label (644,370 150x30), "Auto Mode"
    Lamp1 (788,401 50x50), variable: MAIN.qxEmergySTLamp, style: Lamp-Lamp1-Red
    Label (737,370 150x30), "Emergency Stop"
    Label (456,453 150x30), "Pause"
    Label (555,453 150x30), "Manual"
    Rectangle (157,286 166x30), "%s", text variable: GVL.BufferProducts.Storage1.Component
    Rectangle (348,286 49x30), "%s", text variable: GVL.BufferProducts.Storage1.Quatity
    Rectangle (157,323 166x30), "%s", text variable: GVL.BufferProducts.Storage2.Component
    Rectangle (348,323 49x30), "%s", text variable: GVL.BufferProducts.Storage2.Quatity
    Rectangle (157,360 166x30), "%s", text variable: GVL.BufferProducts.Storage3.Component
    Rectangle (348,360 49x30), "%s", text variable: GVL.BufferProducts.Storage3.Quatity
    PushSwitch (220,201 50x50), behaviour: TAP, style: Switch-PushSwitch-Gray
    PushSwitch (311,202 50x50), behaviour: TAP, style: Switch-PushSwitch-Gray
    PushSwitch (400,200 50x50), behaviour: TAP, style: Switch-PushSwitch-Gray
    Label (165,260 150x30), "Buffer"
    Label (296,260 150x30), "Quantity"
    Label (116,286 37x30), "1"
    Label (116,323 37x30), "2"
    Label (116,361 37x30), "3"
    Rectangle (157,423 166x30), "%s", text variable: MAIN.qsContainer
    Label (165,398 150x30), "Container Color"
    Checkbox (155,462 150x30), "Plate", variable: MAIN.mxPlateAvailable
    Checkbox (155,491 150x30), "Cylinder", variable: MAIN.mxCylinderAvailable
    Checkbox (155,521 150x30), "Octagon", variable: MAIN.mxOctagonAvailable
    GroupBox (121,549 878x300), "Manual Controls"
        Button (14,48 100x30), "Home"
            tap ABB_Control_FB.ixGotoHome
        Button (120,48 100x30), "Scanner"
            tap ABB_Control_FB.ixGotoScanner
        Button (225,48 100x30), "AGV Pos"
            tap ABB_Control_FB.ixGotoAGV
        Button (330,48 100x30), "Buffer"
            tap ABB_Control_FB.ixGotoBuffer
        Button (434,48 100x30), "Table"
            tap ABB_Control_FB.ixGotoTable
        Button (15,119 100x30), "Buffer"
            tap ABB_Control_FB.ixScanBuffer
        Label (95,12 366x30), "Go to Pos"
        Label (95,84 363x30), "Manual Scanning"
        ComboBoxInteger (711,47 150x30), variable: MAIN.mwPartID, text list: MAIN.sPartID
        Label (695,16 182x28), "Part ID"
        Label (518,84 363x30), "Assembling"
        Button (557,118 100x30), "1"
            toggle ABB_Control_FB.ixAssemble1
        Button (40,203 100x30), "Pick"
            tap ABB_Control_FB.ixPickBuffer1
        Button (478,203 100x30), "Pick"
            tap ABB_Control_FB.ixPickAGV
        Button (619,203 100x30), "Pick"
            tap ABB_Control_FB.ixPickScanner
        Button (336,203 100x30), "Pick"
            tap ABB_Control_FB.ixPickBuffer3
        Button (190,203 100x30), "Pick"
            tap ABB_Control_FB.ixPickBuffer2
        Button (39,251 100x30), "Leave"
            tap ABB_Control_FB.ixLeaveBuffer1
        Label (13,168 150x30), "Buffer 1"
        Label (165,168 150x30), "Buffer 2"
        Label (310,168 150x30), "Buffer 3"
        Label (448,169 150x30), "AGV"
        Label (588,168 150x30), "Scanner"
        Label (735,169 150x30), "Table"
        Button (570,18 115x30), "Send Order"
            tap ABB_Control_FB.ixSendOrder
        Button (570,53 115x30), "Finish Order"
            tap ABB_Control_FB.ixFinishOrder
    Label (1062,118 150x30)
    Button (242,668 100x30), "Container"
        tap ABB_Control_FB.ixScanContainer
    Button (347,668 100x30), "Part 1"
        toggle ABB_Control_FB.ixScanPart1
    Button (452,668 100x30), "Part 2"
        toggle ABB_Control_FB.ixScanPart2
    Button (556,668 100x30), "Part 3"
        toggle ABB_Control_FB.ixScanPart3
    Button (783,667 100x30), "2"
        toggle ABB_Control_FB.ixAssemble2
    Button (887,667 100x30), "3"
        toggle ABB_Control_FB.ixAssemble3
    Button (884,752 100x30), "Pick"
        tap ABB_Control_FB.ixPickTable
    Button (598,800 100x30), "Leave"
        tap ABB_Control_FB.ixLeaveAGV
    Button (739,800 100x30), "Leave"
        tap ABB_Control_FB.ixLeaveScanner
    Button (456,800 100x30), "Leave"
        tap ABB_Control_FB.ixLeaveBuffer3
    Button (310,800 100x30), "Leave"
        tap ABB_Control_FB.ixLeaveBuffer2
    Button (883,800 100x30), "Leave"
        tap ABB_Control_FB.ixLeaveTable
END_VISUALIZATION
